TYPE ST_PU_Schuetz_Stellwert :
STRUCT
	Betrieb		: BOOL;
	Freigabe	: BOOL;
END_STRUCT
END_TYPE

(* stored: Version 1.1.0.1, ProductVersion 3.1.4024.9
   DUT ST_PU_Schuetz_Stellwert: Id {28ddfc1b-1401-4e80-9967-203abfce9823} *)
